// SIMATIC S7-200 project (STEP 7-Micro/WIN), CPU 224XP REL 02.01

SYMBOL_TABLE USUARIO1
P_PEATONES       I0.0
C_VERDE          Q0.0
C_AMBAR          Q0.1
C_ROJO           Q0.2
P_ROJO           Q0.3
P_VERDE          Q0.4
SEGURIDAD        Q2.0
END_SYMBOL_TABLE

SYMBOL_TABLE Símbolos S7-200
Primer_ciclo_ON  SM0.1    // ON sólo en el primer ciclo
END_SYMBOL_TABLE

ORGANIZATION_BLOCK PRINCIPAL:OB1
TITLE=COMENTARIOS DEL PROGRAMA
BEGIN
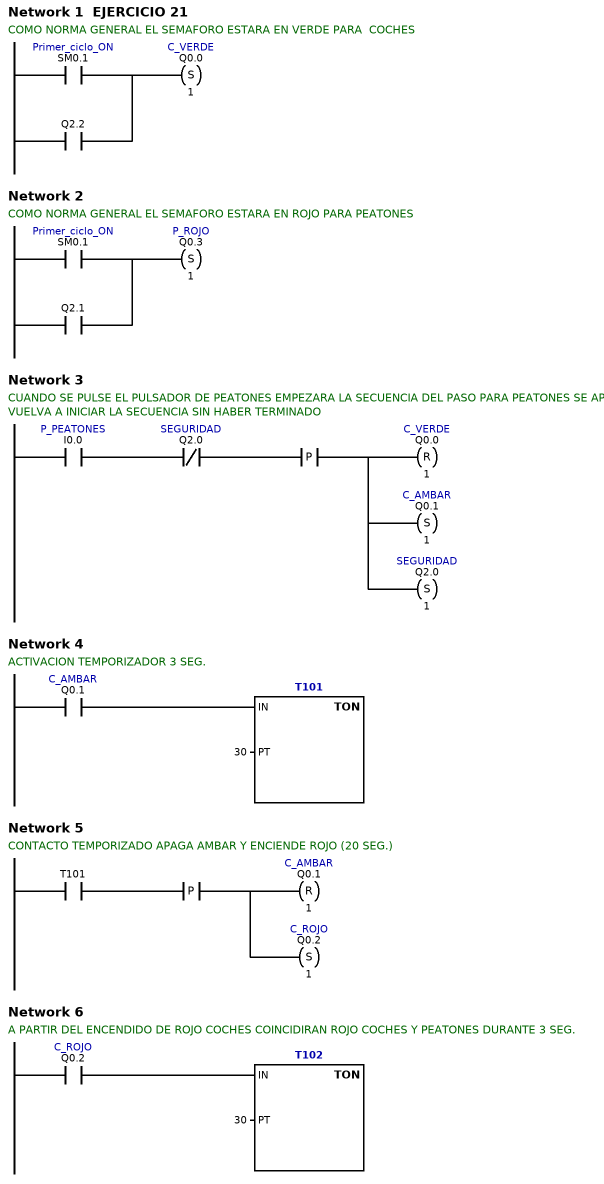
Network 1 // EJERCICIO 21
// COMO NORMA GENERAL EL SEMAFORO ESTARA EN VERDE PARA  COCHES 
LD     Primer_ciclo_ON:SM0.1
O      Q2.2
S      C_VERDE:Q0.0, 1
Network 2
// COMO NORMA GENERAL EL SEMAFORO ESTARA EN ROJO PARA PEATONES
LD     Primer_ciclo_ON:SM0.1
O      Q2.1
S      P_ROJO:Q0.3, 1
Network 3
// CUANDO SE PULSE EL PULSADOR DE PEATONES EMPEZARA LA SECUENCIA DEL PASO PARA PEATONES SE APAGA VERDE COCHES Y SE ENCIENDE AMBAR; MARCA DE SEGUIRIDAD PARA EVITAR QUE VUELVA A INICIAR LA SECUENCIA SIN HABER TERMINADO
LD     P_PEATONES:I0.0
AN     SEGURIDAD:Q2.0
EU
R      C_VERDE:Q0.0, 1
S      C_AMBAR:Q0.1, 1
S      SEGURIDAD:Q2.0, 1
Network 4
// ACTIVACION TEMPORIZADOR 3 SEG.
LD     C_AMBAR:Q0.1
TON    T101, 30
Network 5
// CONTACTO TEMPORIZADO APAGA AMBAR Y ENCIENDE ROJO (20 SEG.)
LD     T101
EU
R      C_AMBAR:Q0.1, 1
S      C_ROJO:Q0.2, 1
Network 6
// A PARTIR DEL ENCENDIDO DE ROJO COCHES COINCIDIRAN ROJO COCHES Y PEATONES DURANTE 3 SEG.
LD     C_ROJO:Q0.2
TON    T102, 30
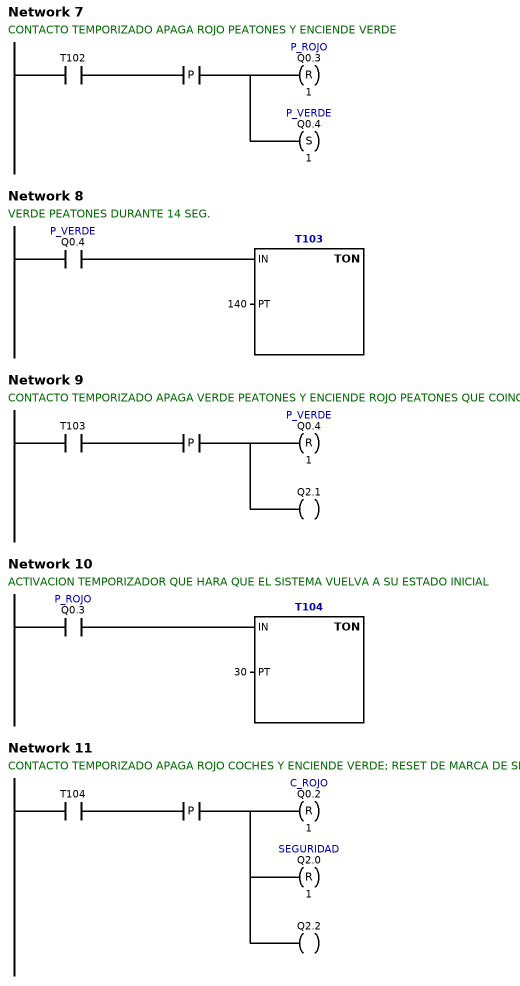
Network 7
// CONTACTO TEMPORIZADO APAGA ROJO PEATONES Y ENCIENDE VERDE
LD     T102
EU
R      P_ROJO:Q0.3, 1
S      P_VERDE:Q0.4, 1
Network 8
// VERDE PEATONES DURANTE 14 SEG. 
LD     P_VERDE:Q0.4
TON    T103, 140
Network 9
// CONTACTO TEMPORIZADO APAGA VERDE PEATONES Y ENCIENDE ROJO PEATONES QUE COINCIDE OTRA VEZ 3 SEG. CON ROJO COCHES
LD     T103
EU
R      P_VERDE:Q0.4, 1
=      Q2.1
Network 10
// ACTIVACION TEMPORIZADOR QUE HARA QUE EL SISTEMA VUELVA A SU ESTADO INICIAL
LD     P_ROJO:Q0.3
TON    T104, 30
Network 11
// CONTACTO TEMPORIZADO APAGA ROJO COCHES Y ENCIENDE VERDE; RESET DE MARCA DE SEGURIDAD PARA PODER INICIAR LA SECUENCIA 
LD     T104
EU
R      C_ROJO:Q0.2, 1
R      SEGURIDAD:Q2.0, 1
=      Q2.2
END_ORGANIZATION_BLOCK
